// TIA Portal V16 export
// export: Created 2024-12-03T15:41:45.4466841Z, ExportSetting WithReadOnly, DisplayName Totally Integrated Automation Portal, DisplayVersion V16 Update 6, DisplayName TIA Portal Version Control Interface, DisplayVersion V16 Update 2, DisplayName TIA Portal Openness, DisplayVersion V16 Update 6, DisplayName TIA Portal Teamcenter Gateway, DisplayVersion V16, DisplayName SINAMICS Startdrive Advanced, DisplayVersion V16 Update 5, DisplayName SINAMICS Startdrive G130, G150, S120, S150, SINAMICS MV, S210, DisplayVersion V16 Update 5, DisplayName SINAMICS Startdrive G110M, G120, G120C, G120D, G120P, G115D, DisplayVersion V16 Update 5, DisplayName STEP 7 Professional, DisplayVersion V16 Update 6, DisplayName STEP 7 Safety, DisplayVersion V16, DisplayName WinCC Advanced / Unified PC, DisplayVersion V16 Update 6
TYPE "G115D_DRIVE_UDT"
// stored: CreationDate 2022-02-10T10:30:20.6863124Z, InterfaceModifiedDate 2021-11-16T12:33:53.9032873Z, IsConsistent true, LibraryConformanceStatus The object is library-conformant., ModifiedDate 2021-11-16T12:33:53.9032873Z
   STRUCT
      Cmd : Struct   // MotorCommands
         Reset : Bool;
         OnAuto : Bool;
         OnManual : Bool;
         DirectionAuto : Bool;
         DirectionManual : Bool;
         SpeedAuto : Real;
         SpeedManual : Real;
         Interlock : Bool;
      END_STRUCT;
      Faults : Struct
         status : Word;
         FaultCode : Word;
         FaultActive : Bool;
         Disconnected : Bool;   // The device is not connected
         TorqueNOK { S7_SetPoint := 'True'} : Bool;
         TemperatureNOK { S7_SetPoint := 'True'} : Bool;
         CurrentNOK { S7_SetPoint := 'True'} : Bool;
         NotOnTImedOut : Bool;   // Motor not on in time
         NotReady : Bool;
         SAFETY_ERROR_ACTIVE : Bool;
         STO_ACTIVE : Bool;
      END_STRUCT;
      Alarms : Struct
         Status : Word;
         AlarmCode : Word;
         AlarmFromDrive : Bool;   // Error from drive
      END_STRUCT;
      Status : Struct
         CmdRunManualActive : Bool;
         Interlocked : Bool;
         ManualModeActive : Bool;
         ManualCommandsDisabled : Bool;
         Running : Bool;
         ActualSpeed : Real;
         ActualDirection : Bool;   // 0 right | 1 left
         Ready : Bool;
         Current : Real;
         Torque : Real;
      END_STRUCT;
      Settings : Struct
         DefaultDirection : Bool;
         AllowManualDirection : Bool;
         MaxSpeedManual : Real := 100.0;
         MinSpeedManual : Real := 0.0;
         MaxSpeedAuto : Real := 100.0;
         MinSpeedAuto : Real := 0.0;
         references : Struct
            maxSpeedReference : Real := 1800.0;
            referenceSpeed : Real := 1500.0;   // rpm
            referenceVoltage : Real := 1000.0;   // Vrms
            referenceCurrent : Real := 100.0;   // Arms
            referenceTorque : Real := 1.0;   // Nm
            referencePower : Real := 0.16;   // Kw
         END_STRUCT;
      END_STRUCT;
      Zone : Int;
      info : "MotorInfo";
   END_STRUCT;
END_TYPE
